PROGRAM MAIN
VAR
  eInit     : e_progress := E_PROGRESS.PROGRESS_DONE;

END_VAR

//############################################################################
// Local time; used for timestamps
//############################################################################
GVL_MSG.fbLocalTime(
                    sLocalTime          => GVL_MSG.sLocalTime, 
                    dtLocalTime         => GVL_MSG.dtLocalTime);

END_PROGRAM

(* stored: Version 1.1.0.1
   POU MAIN: Id {f03fa316-d73a-4a34-ad00-e322fc0b37ed}, SpecialFunc None *)
